PROGRAM P_Modes
VAR
	fbRunning : FB_Running;
END_VAR

fbRunning(
	bAuto := G_Inputs.bAuto,
	bManual := G_Inputs.bManual,
	bStart := G_Inputs.bStartButton,
	bStop := G_Inputs.bStopButton,
	
	bRunning => G_Mode.bRunning,
	bRunning => G_Output.bRunning,
	bManualMode => G_Mode.bManual,
	bAutoMode => G_Mode.bAuto
);

END_PROGRAM

(* stored: Version 1.1.0.1, ProductVersion 3.1.4024.12
   POU P_Modes: Id {022044ba-8743-45e6-a82b-2e81f0455edb}, SpecialFunc None *)
